// TIA Portal V16 export
// export: Created 2021-11-18T22:10:01.724868Z, ExportSetting WithDefaults, DisplayName Totally Integrated Automation Portal, DisplayVersion V16, DisplayName TIA Portal Version Control Interface, DisplayVersion V16, DisplayName TIA Portal Openness, DisplayVersion V16, DisplayName STEP 7 Professional, DisplayVersion V16, DisplayName STEP 7 Safety, DisplayVersion V16, DisplayName WinCC Advanced, DisplayVersion V16
VAR_GLOBAL   // PLC tag table "Default tag table"
   Y1 AT %Q0.0 : Bool;
   Y2 AT %Q0.1 : Bool;
   H1 AT %Q0.2 : Bool;
   H2 AT %Q0.3 : Bool;
   S1 AT %I0.0 : Bool;
   B1 AT %I0.1 : Bool;
   B2 AT %I0.2 : Bool;
   B3 AT %I0.3 : Bool;
   B4 AT %I0.4 : Bool;
   "Step" AT %MW0 : Int;
END_VAR
